TYPE ST105_Fanuc_status_t :
STRUCT
    Picked         : BIT; // Piece(s) picked by the robot
    Placed         : BIT; // Piece(s) placed by the robot
    Ready_to_pick  : BIT; // Robot is in pick position
    Ready_to_place : BIT; // Robot is in place position
    reserve_b4     : BIT; // 
    reserve_b5     : BIT; // 
    reserve_b6     : BIT; // 
    reserve_b7     : BIT; // 
END_STRUCT
END_TYPE

(* stored: Version 1.1.0.1, ProductVersion 3.1.4024.6
   DUT ST105_Fanuc_status_t: Id {b533ae56-77ff-4eff-a336-565c9fd8cfae} *)
